// TIA Portal V18 export
// export: Created 2026-06-09T02:47:52.883472Z, ExportSetting WithDefaults, DisplayName Totally Integrated Automation Portal, DisplayVersion V18, DisplayName TIA Portal Openness, DisplayVersion V18, DisplayName TIA Portal Version Control Interface, DisplayVersion V18, DisplayName STEP 7 Professional, DisplayVersion V18, DisplayName STEP 7 Safety, DisplayVersion V18, DisplayName WinCC Professional, DisplayVersion V18
FUNCTION_BLOCK "Zakrecarka"   // FB2, LAD
{ S7_Optimized_Access := 'TRUE' }
VERSION : 0.1
// stored: AutoNumber true, IsIECCheckEnabled false, IsRetainMemResEnabled false, MemoryReserve 100, SetENOAutomatically false, UDAEnableTagReadback false
   VAR_TEMP   // added for the SCL form of the ladder/FBD networks
      _w1 : Bool;
   END_VAR
BEGIN

REGION Network 1
   // Start przenośnika taśmowego i zapalenie się lampy sygnalizacyjnej.
   // Wyłącznik zakręcarki znajduje się fizycznie na linii produkcyjnej, w jego skład wchodzi również system ryglowania. Stop natomiast w panelu HMI.
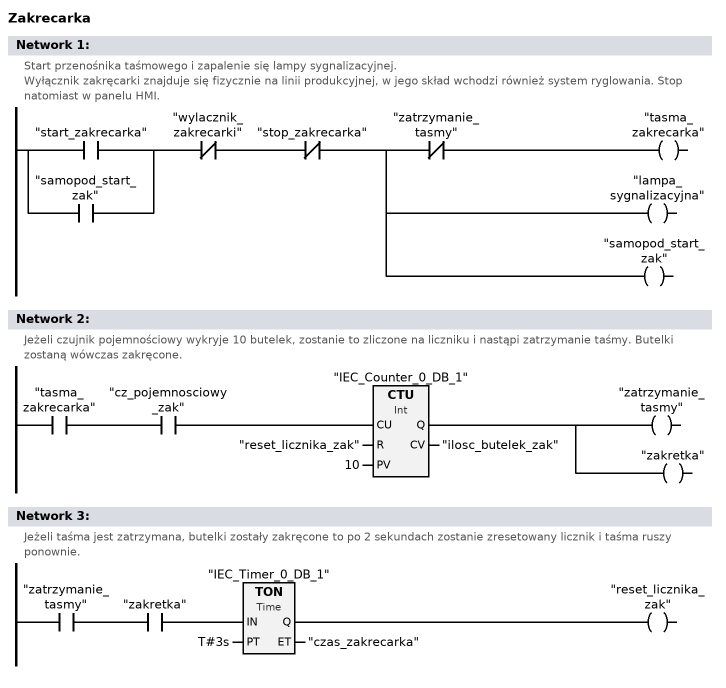
   RUNG wire#powerrail
      Contact( "start_zakrecarka" )
      wire#w1
      I_Contact( "wylacznik_zakrecarki" )
      I_Contact( "stop_zakrecarka" )
      wire#w2
      I_Contact( "zatrzymanie_tasmy" )
      Coil( "tasma_zakrecarka" )
   END_RUNG
   RUNG wire#powerrail
      Contact( "samopod_start_zak" )
   END_RUNG wire#w1
   RUNG wire#w2
      Coil( "lampa_sygnalizacyjna" )
   END_RUNG
   RUNG wire#w2
      Coil( "samopod_start_zak" )
   END_RUNG
   // the same network as SCL:
   #_w1 := ("start_zakrecarka" OR "samopod_start_zak") AND NOT "wylacznik_zakrecarki" AND NOT "stop_zakrecarka";
   "tasma_zakrecarka" := #_w1 AND NOT "zatrzymanie_tasmy";
   "lampa_sygnalizacyjna" := #_w1;
   "samopod_start_zak" := #_w1;
END_REGION

REGION Network 2
   // Jeżeli czujnik pojemnościowy wykryje 10 butelek, zostanie to zliczone na liczniku i nastąpi zatrzymanie taśmy. Butelki zostaną wówczas zakręcone.
   RUNG wire#powerrail
      Contact( "tasma_zakrecarka" )
      Contact( "cz_pojemnosciowy_zak" )
      { S7_Templates := "value_type := Int" } "IEC_Counter_0_DB_1".CTU(r := "reset_licznika_zak", pv := 10, cv => "ilosc_butelek_zak")
      wire#w1
      Coil( "zatrzymanie_tasmy" )
   END_RUNG
   RUNG wire#w1
      Coil( "zakretka" )
   END_RUNG
   // the same network as SCL:
   "IEC_Counter_0_DB_1".CTU(CU := "tasma_zakrecarka" AND "cz_pojemnosciowy_zak",
                           R := "reset_licznika_zak",
                           PV := 10,
                           CV => "ilosc_butelek_zak");
   "zatrzymanie_tasmy" := "IEC_Counter_0_DB_1".Q;
   "zakretka" := "IEC_Counter_0_DB_1".Q;
END_REGION

REGION Network 3
   // Jeżeli taśma jest zatrzymana, butelki zostały zakręcone to po 2 sekundach zostanie zresetowany licznik i taśma ruszy ponownie.
   RUNG wire#powerrail
      Contact( "zatrzymanie_tasmy" )
      Contact( "zakretka" )
      { S7_Templates := "time_type := Time" } "IEC_Timer_0_DB_1".TON(pt := T#3s, et => "czas_zakrecarka")
      Coil( "reset_licznika_zak" )
   END_RUNG
   // the same network as SCL:
   "IEC_Timer_0_DB_1".TON(IN := "zatrzymanie_tasmy" AND "zakretka", PT := T#3s, ET => "czas_zakrecarka");
   "reset_licznika_zak" := "IEC_Timer_0_DB_1".Q;
END_REGION
END_FUNCTION_BLOCK
